PROGRAM P_Demo_FB_DALIV2StepUp
VAR
    fbFB_DALIV2StepUp        : FB_DALIV2StepUp;
    stCommandBuffer : ST_DALIV2CommandBuffer;

    bTrigger        : BOOL;
    nLampAddr        : BYTE := 0;


    bBusy           : BOOL;
    bErr            : BOOL;
    nErrId          : UDINT;
END_VAR

// =============================================================================
// 场景：面板长按加亮按钮：每 100 ms 触发一次本 FB。...
//
// 价值：DALI 协议标准命令的轻量封装。
//
// 验证步骤：
//   1. 通信 FB 跑起；编译；登录。
//   2. 在线 bTrigger 一次上升沿；等 bBusy 回 FALSE。
//   3. 观察 short addr 0 灯的物理亮度变化是否符合本命令描述。
// =============================================================================
fbFB_DALIV2StepUp(
    bStart           := bTrigger,
    nAddr            := nLampAddr,
    eAddrType        := eDALIV2AddrTypeShort,
    eCommandPriority := eDALIV2CommandPriorityMiddle,
    stCommandBuffer  := stCommandBuffer
);

bBusy  := fbFB_DALIV2StepUp.bBusy;
bErr   := fbFB_DALIV2StepUp.bError;
nErrId := fbFB_DALIV2StepUp.nErrorId;

END_PROGRAM

(* stored: Version 1.1.0.1, ProductVersion 3.1.4024.5
   POU P_Demo_FB_DALIV2StepUp: Id {83061058-10cd-5f3a-a69b-eef3c6df802c}, SpecialFunc None *)
